LIN {E6POS: X 1455.051, Y -12.200, Z 516.145, A 42.957, B 70.046, C -138.807, E1 0.000, E2 0.0, E3 0.0, E4 0.0, E5 0.0, E6 0.0} C_DIS
;POWDER FEED RATE  =  3.0
;LASER INTENSITY  =  4.0
LIN {E6POS: X 1445.585, Y -2.040, Z 516.145, A 43.012, B 69.711, C -138.813, E1 0.000, E2 0.0, E3 0.0, E4 0.0, E5 0.0, E6 0.0} C_DIS
;POWDER FEED RATE  =  3.0
;LASER INTENSITY  =  4.0
LIN {E6POS: X 1436.083, Y 8.120, Z 516.145, A 43.176, B 69.386, C -138.711, E1 0.000, E2 0.0, E3 0.0, E4 0.0, E5 0.0, E6 0.0} C_DIS
;POWDER FEED RATE  =  3.0
;LASER INTENSITY  =  4.0
LIN {E6POS: X 1426.508, Y 18.280, Z 516.145, A 43.446, B 69.128, C -138.490, E1 0.000, E2 0.0, E3 0.0, E4 0.0, E5 0.0, E6 0.0} C_DIS
;POWDER FEED RATE  =  3.0
;LASER INTENSITY  =  4.0
LIN {E6POS: X 1417.104, Y 28.440, Z 516.393, A 48.821, B 67.331, C -133.472, E1 0.000, E2 0.0, E3 0.0, E4 0.0, E5 0.0, E6 0.0} C_DIS
;POWDER FEED RATE  =  3.0
;LASER INTENSITY  =  4.0
LIN {E6POS: X 1409.237, Y 38.600, Z 518.129, A 60.642, B 62.204, C -122.451, E1 0.000, E2 0.0, E3 0.0, E4 0.0, E5 0.0, E6 0.0} C_DIS
;POWDER FEED RATE  =  3.0
;LASER INTENSITY  =  4.0
LIN {E6POS: X 1404.551, Y 48.760, Z 522.839, A 72.980, B 53.267, C -110.905, E1 0.000, E2 0.0, E3 0.0, E4 0.0, E5 0.0, E6 0.0} C_DIS
;POWDER FEED RATE  =  3.0
;LASER INTENSITY  =  4.0
LIN {E6POS: X 1403.886, Y 58.920, Z 531.268, A 80.416, B 46.343, C -103.137, E1 0.000, E2 0.0, E3 0.0, E4 0.0, E5 0.0, E6 0.0} C_DIS
;POWDER FEED RATE  =  3.0
;LASER INTENSITY  =  4.0
LIN {E6POS: X 1404.867, Y 69.080, Z 541.185, A 83.811, B 46.478, C -98.506, E1 0.000, E2 0.0, E3 0.0, E4 0.0, E5 0.0, E6 0.0} C_DIS
;POWDER FEED RATE  =  3.0
;LASER INTENSITY  =  4.0
LIN {E6POS: X 1404.312, Y 79.240, Z 549.614, A 84.676, B 55.923, C -96.419, E1 0.000, E2 0.0, E3 0.0, E4 0.0, E5 0.0, E6 0.0} C_DIS
;POWDER FEED RATE  =  3.0
;LASER INTENSITY  =  4.0
LIN {E6POS: X 1399.832, Y 89.400, Z 554.324, A 82.280, B 72.116, C -98.107, E1 0.000, E2 0.0, E3 0.0, E4 0.0, E5 0.0, E6 0.0} C_DIS
;POWDER FEED RATE  =  3.0
;LASER INTENSITY  =  4.0
LIN {E6POS: X 1392.206, Y 99.560, Z 556.059, A 70.618, B 83.671, C -109.492, E1 0.000, E2 0.0, E3 0.0, E4 0.0, E5 0.0, E6 0.0} C_DIS
;POWDER FEED RATE  =  3.0
;LASER INTENSITY  =  4.0
LIN {E6POS: X 1383.008, Y 109.720, Z 556.307, A 42.957, B 87.164, C -137.078, E1 0.000, E2 0.0, E3 0.0, E4 0.0, E5 0.0, E6 0.0} C_DIS
;POWDER FEED RATE  =  3.0
;LASER INTENSITY  =  4.0
LIN {E6POS: X 1373.548, Y 119.880, Z 556.307, A 42.957, B 87.129, C -137.079, E1 0.000, E2 0.0, E3 0.0, E4 0.0, E5 0.0, E6 0.0} C_DIS
;POWDER FEED RATE  =  3.0
;LASER INTENSITY  =  4.0
LIN {E6POS: X 1364.087, Y 130.040, Z 556.307, A 42.957, B 87.094, C -137.079, E1 0.000, E2 0.0, E3 0.0, E4 0.0, E5 0.0, E6 0.0} C_DIS
;POWDER FEED RATE  =  3.0
;LASER INTENSITY  =  4.0
LIN {E6POS: X 1354.627, Y 140.200, Z 556.307, A 42.957, B 87.057, C -137.080, E1 0.000, E2 0.0, E3 0.0, E4 0.0, E5 0.0, E6 0.0} C_DIS
;POWDER FEED RATE  =  3.0
;LASER INTENSITY  =  4.0
>>>>>>>>>>>>>>>>>>>>>>>>>>>>POWDER FEED OFF  at=START
>>>>>>>>>>>>>>>>>>>>>>>>>>>>LASER OFF at=START
>>>>>>>>>>>>>>>>>>>>>>>>>>>>GAS SUPPLY OFF  at=START
LIN {E6POS: X 1354.627, Y 140.200, Z 556.307, A 42.957, B 87.057, C -137.080, E1 0.000, E2 0.0, E3 0.0, E4 0.0, E5 0.0, E6 0.0} C_DIS
LIN {E6POS: X 1364.087, Y 130.040, Z 556.307, A 42.957, B 87.094, C -137.079, E1 0.000, E2 0.0, E3 0.0, E4 0.0, E5 0.0, E6 0.0} C_DIS
LIN {E6POS: X 1364.087, Y 130.040, Z 556.307, A 42.957, B 87.094, C -137.079, E1 0.000, E2 0.0, E3 0.0, E4 0.0, E5 0.0, E6 0.0} C_DIS
>>>>>>>>>>>>>>>>>>>>>>>>>>>>GAS SUPPLY ON at=END
>>>>>>>>>>>>>>>>>>>>>>>>>>>>POWDER FEED ON at=END
>>>>>>>>>>>>>>>>>>>>>>>>>>>>LASER ON at=END
LIN {E6POS: X 1459.969, Y -12.200, Z 517.448, A 43.187, B 70.234, C -138.545, E1 0.000, E2 0.0, E3 0.0, E4 0.0, E5 0.0, E6 0.0} C_DIS
;POWDER FEED RATE  =  3.0
;LASER INTENSITY  =  4.0
LIN {E6POS: X 1450.428, Y -2.040, Z 517.448, A 43.224, B 69.979, C -138.554, E1 0.000, E2 0.0, E3 0.0, E4 0.0, E5 0.0, E6 0.0} C_DIS
;POWDER FEED RATE  =  3.0
;LASER INTENSITY  =  4.0
LIN {E6POS: X 1440.864, Y 8.120, Z 517.448, A 43.333, B 69.736, C -138.490, E1 0.000, E2 0.0, E3 0.0, E4 0.0, E5 0.0, E6 0.0} C_DIS
;POWDER FEED RATE  =  3.0
;LASER INTENSITY  =  4.0
LIN {E6POS: X 1431.250, Y 18.280, Z 517.448, A 43.513, B 69.549, C -138.345, E1 0.000, E2 0.0, E3 0.0, E4 0.0, E5 0.0, E6 0.0} C_DIS
;POWDER FEED RATE  =  3.0
;LASER INTENSITY  =  4.0
LIN {E6POS: X 1421.855, Y 28.440, Z 517.689, A 48.669, B 67.874, C -133.513, E1 0.000, E2 0.0, E3 0.0, E4 0.0, E5 0.0, E6 0.0} C_DIS
;POWDER FEED RATE  =  3.0
;LASER INTENSITY  =  4.0
LIN {E6POS: X 1414.112, Y 38.600, Z 519.378, A 60.307, B 63.006, C -122.617, E1 0.000, E2 0.0, E3 0.0, E4 0.0, E5 0.0, E6 0.0} C_DIS
;POWDER FEED RATE  =  3.0
;LASER INTENSITY  =  4.0
LIN {E6POS: X 1409.744, Y 48.760, Z 523.963, A 72.750, B 54.338, C -110.916, E1 0.000, E2 0.0, E3 0.0, E4 0.0, E5 0.0, E6 0.0} C_DIS
;POWDER FEED RATE  =  3.0
;LASER INTENSITY  =  4.0
LIN {E6POS: X 1409.627, Y 58.920, Z 532.166, A 80.409, B 47.407, C -102.927, E1 0.000, E2 0.0, E3 0.0, E4 0.0, E5 0.0, E6 0.0} C_DIS
;POWDER FEED RATE  =  3.0
;LASER INTENSITY  =  4.0
LIN {E6POS: X 1411.234, Y 69.080, Z 541.818, A 83.997, B 47.432, C -98.125, E1 0.000, E2 0.0, E3 0.0, E4 0.0, E5 0.0, E6 0.0} C_DIS
;POWDER FEED RATE  =  3.0
;LASER INTENSITY  =  4.0
LIN {E6POS: X 1411.190, Y 79.240, Z 550.021, A 85.122, B 56.795, C -95.824, E1 0.000, E2 0.0, E3 0.0, E4 0.0, E5 0.0, E6 0.0} C_DIS
;POWDER FEED RATE  =  3.0
;LASER INTENSITY  =  4.0
LIN {E6POS: X 1406.961, Y 89.400, Z 554.606, A 83.358, B 72.840, C -96.948, E1 0.000, E2 0.0, E3 0.0, E4 0.0, E5 0.0, E6 0.0} C_DIS
;POWDER FEED RATE  =  3.0
;LASER INTENSITY  =  4.0
LIN {E6POS: X 1399.379, Y 99.560, Z 556.295, A 73.249, B 84.276, C -106.830, E1 0.000, E2 0.0, E3 0.0, E4 0.0, E5 0.0, E6 0.0} C_DIS
;POWDER FEED RATE  =  3.0
;LASER INTENSITY  =  4.0
LIN {E6POS: X 1390.122, Y 109.720, Z 556.536, A 43.187, B 87.789, C -136.834, E1 0.000, E2 0.0, E3 0.0, E4 0.0, E5 0.0, E6 0.0} C_DIS
;POWDER FEED RATE  =  3.0
;LASER INTENSITY  =  4.0
LIN {E6POS: X 1380.585, Y 119.880, Z 556.536, A 43.187, B 87.769, C -136.834, E1 0.000, E2 0.0, E3 0.0, E4 0.0, E5 0.0, E6 0.0} C_DIS
;POWDER FEED RATE  =  3.0
;LASER INTENSITY  =  4.0
LIN {E6POS: X 1371.049, Y 130.040, Z 556.536, A 43.187, B 87.747, C -136.835, E1 0.000, E2 0.0, E3 0.0, E4 0.0, E5 0.0, E6 0.0} C_DIS
;POWDER FEED RATE  =  3.0
;LASER INTENSITY  =  4.0
LIN {E6POS: X 1361.512, Y 140.200, Z 556.536, A 43.187, B 87.725, C -136.835, E1 0.000, E2 0.0, E3 0.0, E4 0.0, E5 0.0, E6 0.0} C_DIS
;POWDER FEED RATE  =  3.0
;LASER INTENSITY  =  4.0
>>>>>>>>>>>>>>>>>>>>>>>>>>>>POWDER FEED OFF  at=START
>>>>>>>>>>>>>>>>>>>>>>>>>>>>LASER OFF at=START
>>>>>>>>>>>>>>>>>>>>>>>>>>>>GAS SUPPLY OFF  at=START
LIN {E6POS: X 1361.512, Y 140.200, Z 556.536, A 43.187, B 87.725, C -136.835, E1 0.000, E2 0.0, E3 0.0, E4 0.0, E5 0.0, E6 0.0} C_DIS
LIN {E6POS: X 1371.049, Y 130.040, Z 556.536, A 43.187, B 87.747, C -136.835, E1 0.000, E2 0.0, E3 0.0, E4 0.0, E5 0.0, E6 0.0} C_DIS
LIN {E6POS: X 1371.049, Y 130.040, Z 556.536, A 43.187, B 87.747, C -136.835, E1 0.000, E2 0.0, E3 0.0, E4 0.0, E5 0.0, E6 0.0} C_DIS
>>>>>>>>>>>>>>>>>>>>>>>>>>>>GAS SUPPLY ON at=END
>>>>>>>>>>>>>>>>>>>>>>>>>>>>POWDER FEED ON at=END
>>>>>>>>>>>>>>>>>>>>>>>>>>>>LASER ON at=END
LIN {E6POS: X 1464.867, Y -12.200, Z 518.698, A 43.359, B 71.280, C -138.192, E1 0.000, E2 0.0, E3 0.0, E4 0.0, E5 0.0, E6 0.0} C_DIS
;POWDER FEED RATE  =  3.0
;LASER INTENSITY  =  4.0
LIN {E6POS: X 1455.270, Y -2.040, Z 518.698, A 43.382, B 71.104, C -138.200, E1 0.000, E2 0.0, E3 0.0, E4 0.0, E5 0.0, E6 0.0} C_DIS
;POWDER FEED RATE  =  3.0
;LASER INTENSITY  =  4.0
LIN {E6POS: X 1445.658, Y 8.120, Z 518.698, A 43.450, B 70.939, C -138.160, E1 0.000, E2 0.0, E3 0.0, E4 0.0, E5 0.0, E6 0.0} C_DIS
;POWDER FEED RATE  =  3.0
;LASER INTENSITY  =  4.0
LIN {E6POS: X 1436.016, Y 18.280, Z 518.698, A 43.563, B 70.815, C -138.068, E1 0.000, E2 0.0, E3 0.0, E4 0.0, E5 0.0, E6 0.0} C_DIS
;POWDER FEED RATE  =  3.0
;LASER INTENSITY  =  4.0
LIN {E6POS: X 1426.630, Y 28.440, Z 518.932, A 48.837, B 69.183, C -133.087, E1 0.000, E2 0.0, E3 0.0, E4 0.0, E5 0.0, E6 0.0} C_DIS
;POWDER FEED RATE  =  3.0
;LASER INTENSITY  =  4.0
LIN {E6POS: X 1419.000, Y 38.600, Z 520.575, A 60.708, B 64.304, C -121.904, E1 0.000, E2 0.0, E3 0.0, E4 0.0, E5 0.0, E6 0.0} C_DIS
;POWDER FEED RATE  =  3.0
;LASER INTENSITY  =  4.0
LIN {E6POS: X 1414.928, Y 48.760, Z 525.033, A 73.166, B 55.549, C -110.150, E1 0.000, E2 0.0, E3 0.0, E4 0.0, E5 0.0, E6 0.0} C_DIS
;POWDER FEED RATE  =  3.0
;LASER INTENSITY  =  4.0
LIN {E6POS: X 1415.321, Y 58.920, Z 533.010, A 80.752, B 48.468, C -102.271, E1 0.000, E2 0.0, E3 0.0, E4 0.0, E5 0.0, E6 0.0} C_DIS
;POWDER FEED RATE  =  3.0
;LASER INTENSITY  =  4.0
LIN {E6POS: X 1417.517, Y 69.080, Z 542.395, A 84.350, B 48.378, C -97.539, E1 0.000, E2 0.0, E3 0.0, E4 0.0, E5 0.0, E6 0.0} C_DIS
;POWDER FEED RATE  =  3.0
;LASER INTENSITY  =  4.0
LIN {E6POS: X 1417.956, Y 79.240, Z 550.373, A 85.638, B 57.664, C -95.159, E1 0.000, E2 0.0, E3 0.0, E4 0.0, E5 0.0, E6 0.0} C_DIS
;POWDER FEED RATE  =  3.0
;LASER INTENSITY  =  4.0
LIN {E6POS: X 1413.970, Y 89.400, Z 554.831, A 84.454, B 73.537, C -95.781, E1 0.000, E2 0.0, E3 0.0, E4 0.0, E5 0.0, E6 0.0} C_DIS
;POWDER FEED RATE  =  3.0
;LASER INTENSITY  =  4.0
LIN {E6POS: X 1406.442, Y 99.560, Z 556.473, A 76.097, B 84.824, C -103.958, E1 0.000, E2 0.0, E3 0.0, E4 0.0, E5 0.0, E6 0.0} C_DIS
;POWDER FEED RATE  =  3.0
;LASER INTENSITY  =  4.0
LIN {E6POS: X 1397.144, Y 109.720, Z 556.708, A 43.359, B 88.351, C -136.653, E1 0.000, E2 0.0, E3 0.0, E4 0.0, E5 0.0, E6 0.0} C_DIS
;POWDER FEED RATE  =  3.0
;LASER INTENSITY  =  4.0
LIN {E6POS: X 1387.550, Y 119.880, Z 556.708, A 43.359, B 88.339, C -136.653, E1 0.000, E2 0.0, E3 0.0, E4 0.0, E5 0.0, E6 0.0} C_DIS
;POWDER FEED RATE  =  3.0
;LASER INTENSITY  =  4.0
LIN {E6POS: X 1377.956, Y 130.040, Z 556.708, A 43.359, B 88.328, C -136.653, E1 0.000, E2 0.0, E3 0.0, E4 0.0, E5 0.0, E6 0.0} C_DIS
;POWDER FEED RATE  =  3.0
;LASER INTENSITY  =  4.0
LIN {E6POS: X 1368.361, Y 140.200, Z 556.708, A 43.359, B 88.316, C -136.653, E1 0.000, E2 0.0, E3 0.0, E4 0.0, E5 0.0, E6 0.0} C_DIS
;POWDER FEED RATE  =  3.0
;LASER INTENSITY  =  4.0
>>>>>>>>>>>>>>>>>>>>>>>>>>>>POWDER FEED OFF  at=START
>>>>>>>>>>>>>>>>>>>>>>>>>>>>LASER OFF at=START
>>>>>>>>>>>>>>>>>>>>>>>>>>>>GAS SUPPLY OFF  at=START
LIN {E6POS: X 1368.361, Y 140.200, Z 556.708, A 43.359, B 88.316, C -136.653, E1 0.000, E2 0.0, E3 0.0, E4 0.0, E5 0.0, E6 0.0} C_DIS
LIN {E6POS: X 1377.956, Y 130.040, Z 556.708, A 43.359, B 88.328, C -136.653, E1 0.000, E2 0.0, E3 0.0, E4 0.0, E5 0.0, E6 0.0} C_DIS
LIN {E6POS: X 1377.956, Y 130.040, Z 556.708, A 43.359, B 88.328, C -136.653, E1 0.000, E2 0.0, E3 0.0, E4 0.0, E5 0.0, E6 0.0} C_DIS
>>>>>>>>>>>>>>>>>>>>>>>>>>>>GAS SUPPLY ON at=END
>>>>>>>>>>>>>>>>>>>>>>>>>>>>POWDER FEED ON at=END
>>>>>>>>>>>>>>>>>>>>>>>>>>>>LASER ON at=END
LIN {E6POS: X 1469.825, Y -12.200, Z 519.857, A 43.481, B 73.154, C -137.772, E1 0.000, E2 0.0, E3 0.0, E4 0.0, E5 0.0, E6 0.0} C_DIS
;POWDER FEED RATE  =  3.0
;LASER INTENSITY  =  4.0
LIN {E6POS: X 1460.188, Y -2.040, Z 519.857, A 43.494, B 73.045, C -137.775, E1 0.000, E2 0.0, E3 0.0, E4 0.0, E5 0.0, E6 0.0} C_DIS
;POWDER FEED RATE  =  3.0
;LASER INTENSITY  =  4.0
LIN {E6POS: X 1450.543, Y 8.120, Z 519.857, A 43.534, B 72.945, C -137.751, E1 0.000, E2 0.0, E3 0.0, E4 0.0, E5 0.0, E6 0.0} C_DIS
;POWDER FEED RATE  =  3.0
;LASER INTENSITY  =  4.0
LIN {E6POS: X 1440.880, Y 18.280, Z 519.857, A 43.599, B 72.872, C -137.697, E1 0.000, E2 0.0, E3 0.0, E4 0.0, E5 0.0, E6 0.0} C_DIS
;POWDER FEED RATE  =  3.0
;LASER INTENSITY  =  4.0
LIN {E6POS: X 1431.504, Y 28.440, Z 520.085, A 49.405, B 71.202, C -132.153, E1 0.000, E2 0.0, E3 0.0, E4 0.0, E5 0.0, E6 0.0} C_DIS
;POWDER FEED RATE  =  3.0
;LASER INTENSITY  =  4.0
LIN {E6POS: X 1423.975, Y 38.600, Z 521.683, A 61.989, B 66.034, C -120.206, E1 0.000, E2 0.0, E3 0.0, E4 0.0, E5 0.0, E6 0.0} C_DIS
;POWDER FEED RATE  =  3.0
;LASER INTENSITY  =  4.0
LIN {E6POS: X 1420.168, Y 48.760, Z 526.019, A 74.316, B 56.821, C -108.546, E1 0.000, E2 0.0, E3 0.0, E4 0.0, E5 0.0, E6 0.0} C_DIS
;POWDER FEED RATE  =  3.0
;LASER INTENSITY  =  4.0
LIN {E6POS: X 1421.025, Y 58.920, Z 533.779, A 81.485, B 49.455, C -101.145, E1 0.000, E2 0.0, E3 0.0, E4 0.0, E5 0.0, E6 0.0} C_DIS
;POWDER FEED RATE  =  3.0
;LASER INTENSITY  =  4.0
LIN {E6POS: X 1423.755, Y 69.080, Z 542.909, A 84.887, B 49.265, C -96.735, E1 0.000, E2 0.0, E3 0.0, E4 0.0, E5 0.0, E6 0.0} C_DIS
;POWDER FEED RATE  =  3.0
;LASER INTENSITY  =  4.0
LIN {E6POS: X 1424.638, Y 79.240, Z 550.669, A 86.227, B 58.494, C -94.423, E1 0.000, E2 0.0, E3 0.0, E4 0.0, E5 0.0, E6 0.0} C_DIS
;POWDER FEED RATE  =  3.0
;LASER INTENSITY  =  4.0
LIN {E6POS: X 1420.881, Y 89.400, Z 555.005, A 85.552, B 74.187, C -94.622, E1 0.000, E2 0.0, E3 0.0, E4 0.0, E5 0.0, E6 0.0} C_DIS
;POWDER FEED RATE  =  3.0
;LASER INTENSITY  =  4.0
LIN {E6POS: X 1413.412, Y 99.560, Z 556.603, A 79.104, B 85.302, C -100.932, E1 0.000, E2 0.0, E3 0.0, E4 0.0, E5 0.0, E6 0.0} C_DIS
;POWDER FEED RATE  =  3.0
;LASER INTENSITY  =  4.0
LIN {E6POS: X 1404.086, Y 109.720, Z 556.831, A 43.481, B 88.840, C -136.525, E1 0.000, E2 0.0, E3 0.0, E4 0.0, E5 0.0, E6 0.0} C_DIS
;POWDER FEED RATE  =  3.0
;LASER INTENSITY  =  4.0
LIN {E6POS: X 1394.451, Y 119.880, Z 556.831, A 43.481, B 88.835, C -136.525, E1 0.000, E2 0.0, E3 0.0, E4 0.0, E5 0.0, E6 0.0} C_DIS
;POWDER FEED RATE  =  3.0
;LASER INTENSITY  =  4.0
LIN {E6POS: X 1384.816, Y 130.040, Z 556.831, A 43.481, B 88.829, C -136.525, E1 0.000, E2 0.0, E3 0.0, E4 0.0, E5 0.0, E6 0.0} C_DIS
;POWDER FEED RATE  =  3.0
;LASER INTENSITY  =  4.0
LIN {E6POS: X 1375.181, Y 140.200, Z 556.831, A 43.481, B 88.823, C -136.525, E1 0.000, E2 0.0, E3 0.0, E4 0.0, E5 0.0, E6 0.0} C_DIS
;POWDER FEED RATE  =  3.0
;LASER INTENSITY  =  4.0
>>>>>>>>>>>>>>>>>>>>>>>>>>>>POWDER FEED OFF  at=START
>>>>>>>>>>>>>>>>>>>>>>>>>>>>LASER OFF at=START
>>>>>>>>>>>>>>>>>>>>>>>>>>>>GAS SUPPLY OFF  at=START
LIN {E6POS: X 1375.181, Y 140.200, Z 556.831, A 43.481, B 88.823, C -136.525, E1 0.000, E2 0.0, E3 0.0, E4 0.0, E5 0.0, E6 0.0} C_DIS
LIN {E6POS: X 1384.816, Y 130.040, Z 556.831, A 43.481, B 88.829, C -136.525, E1 0.000, E2 0.0, E3 0.0, E4 0.0, E5 0.0, E6 0.0} C_DIS
LIN {E6POS: X 1384.816, Y 130.040, Z 556.831, A 43.481, B 88.829, C -136.525, E1 0.000, E2 0.0, E3 0.0, E4 0.0, E5 0.0, E6 0.0} C_DIS
>>>>>>>>>>>>>>>>>>>>>>>>>>>>GAS SUPPLY ON at=END
>>>>>>>>>>>>>>>>>>>>>>>>>>>>POWDER FEED ON at=END
>>>>>>>>>>>>>>>>>>>>>>>>>>>>LASER ON at=END
LIN {E6POS: X 1474.925, Y -12.200, Z 520.889, A 43.563, B 75.759, C -137.329, E1 0.000, E2 0.0, E3 0.0, E4 0.0, E5 0.0, E6 0.0} C_DIS
;POWDER FEED RATE  =  3.0
;LASER INTENSITY  =  4.0
LIN {E6POS: X 1465.262, Y -2.040, Z 520.889, A 43.570, B 75.702, C -137.330, E1 0.000, E2 0.0, E3 0.0, E4 0.0, E5 0.0, E6 0.0} C_DIS
;POWDER FEED RATE  =  3.0
;LASER INTENSITY  =  4.0
LIN {E6POS: X 1455.594, Y 8.120, Z 520.889, A 43.590, B 75.650, C -137.316, E1 0.000, E2 0.0, E3 0.0, E4 0.0, E5 0.0, E6 0.0} C_DIS
;POWDER FEED RATE  =  3.0
;LASER INTENSITY  =  4.0
LIN {E6POS: X 1445.917, Y 18.280, Z 520.889, A 43.623, B 75.613, C -137.287, E1 0.000, E2 0.0, E3 0.0, E4 0.0, E5 0.0, E6 0.0} C_DIS
;POWDER FEED RATE  =  3.0
;LASER INTENSITY  =  4.0
LIN {E6POS: X 1436.550, Y 28.440, Z 521.112, A 50.550, B 73.825, C -130.590, E1 0.000, E2 0.0, E3 0.0, E4 0.0, E5 0.0, E6 0.0} C_DIS
;POWDER FEED RATE  =  3.0
;LASER INTENSITY  =  4.0
LIN {E6POS: X 1429.109, Y 38.600, Z 522.668, A 64.346, B 68.087, C -117.369, E1 0.000, E2 0.0, E3 0.0, E4 0.0, E5 0.0, E6 0.0} C_DIS
;POWDER FEED RATE  =  3.0
;LASER INTENSITY  =  4.0
LIN {E6POS: X 1425.532, Y 48.760, Z 526.893, A 76.244, B 58.061, C -106.091, E1 0.000, E2 0.0, E3 0.0, E4 0.0, E5 0.0, E6 0.0} C_DIS
;POWDER FEED RATE  =  3.0
;LASER INTENSITY  =  4.0
LIN {E6POS: X 1426.793, Y 58.920, Z 534.454, A 82.621, B 50.297, C -99.555, E1 0.000, E2 0.0, E3 0.0, E4 0.0, E5 0.0, E6 0.0} C_DIS
;POWDER FEED RATE  =  3.0
;LASER INTENSITY  =  4.0
LIN {E6POS: X 1429.992, Y 69.080, Z 543.349, A 85.614, B 50.041, C -95.714, E1 0.000, E2 0.0, E3 0.0, E4 0.0, E5 0.0, E6 0.0} C_DIS
;POWDER FEED RATE  =  3.0
;LASER INTENSITY  =  4.0
LIN {E6POS: X 1431.266, Y 79.240, Z 550.909, A 86.889, B 59.250, C -93.619, E1 0.000, E2 0.0, E3 0.0, E4 0.0, E5 0.0, E6 0.0} C_DIS
;POWDER FEED RATE  =  3.0
;LASER INTENSITY  =  4.0
LIN {E6POS: X 1427.715, Y 89.400, Z 555.134, A 86.628, B 74.770, C -93.495, E1 0.000, E2 0.0, E3 0.0, E4 0.0, E5 0.0, E6 0.0} C_DIS
;POWDER FEED RATE  =  3.0
;LASER INTENSITY  =  4.0
LIN {E6POS: X 1420.304, Y 99.560, Z 556.691, A 82.147, B 85.702, C -97.875, E1 0.000, E2 0.0, E3 0.0, E4 0.0, E5 0.0, E6 0.0} C_DIS
;POWDER FEED RATE  =  3.0
;LASER INTENSITY  =  4.0
LIN {E6POS: X 1410.963, Y 109.720, Z 556.913, A 43.563, B 89.250, C -136.439, E1 0.000, E2 0.0, E3 0.0, E4 0.0, E5 0.0, E6 0.0} C_DIS
;POWDER FEED RATE  =  3.0
;LASER INTENSITY  =  4.0
LIN {E6POS: X 1401.300, Y 119.880, Z 556.913, A 43.563, B 89.248, C -136.439, E1 0.000, E2 0.0, E3 0.0, E4 0.0, E5 0.0, E6 0.0} C_DIS
;POWDER FEED RATE  =  3.0
;LASER INTENSITY  =  4.0
LIN {E6POS: X 1391.638, Y 130.040, Z 556.913, A 43.563, B 89.246, C -136.439, E1 0.000, E2 0.0, E3 0.0, E4 0.0, E5 0.0, E6 0.0} C_DIS
;POWDER FEED RATE  =  3.0
;LASER INTENSITY  =  4.0
LIN {E6POS: X 1381.975, Y 140.200, Z 556.913, A 43.563, B 89.243, C -136.439, E1 0.000, E2 0.0, E3 0.0, E4 0.0, E5 0.0, E6 0.0} C_DIS
;POWDER FEED RATE  =  3.0
;LASER INTENSITY  =  4.0
>>>>>>>>>>>>>>>>>>>>>>>>>>>>POWDER FEED OFF  at=START
>>>>>>>>>>>>>>>>>>>>>>>>>>>>LASER OFF at=START
>>>>>>>>>>>>>>>>>>>>>>>>>>>>GAS SUPPLY OFF  at=START
LIN {E6POS: X 1381.975, Y 140.200, Z 556.913, A 43.563, B 89.243, C -136.439, E1 0.000, E2 0.0, E3 0.0, E4 0.0, E5 0.0, E6 0.0} C_DIS
LIN {E6POS: X 1391.638, Y 130.040, Z 556.913, A 43.563, B 89.246, C -136.439, E1 0.000, E2 0.0, E3 0.0, E4 0.0, E5 0.0, E6 0.0} C_DIS
LIN {E6POS: X 1391.638, Y 130.040, Z 556.913, A 43.563, B 89.246, C -136.439, E1 0.000, E2 0.0, E3 0.0, E4 0.0, E5 0.0, E6 0.0} C_DIS
>>>>>>>>>>>>>>>>>>>>>>>>>>>>GAS SUPPLY ON at=END
>>>>>>>>>>>>>>>>>>>>>>>>>>>>POWDER FEED ON at=END
>>>>>>>>>>>>>>>>>>>>>>>>>>>>LASER ON at=END
LIN {E6POS: X 1480.249, Y -12.200, Z 521.757, A 43.613, B 78.943, C -136.923, E1 0.000, E2 0.0, E3 0.0, E4 0.0, E5 0.0, E6 0.0} C_DIS
;POWDER FEED RATE  =  3.0
;LASER INTENSITY  =  4.0
LIN {E6POS: X 1470.570, Y -2.040, Z 521.757, A 43.615, B 78.919, C -136.923, E1 0.000, E2 0.0, E3 0.0, E4 0.0, E5 0.0, E6 0.0} C_DIS
;POWDER FEED RATE  =  3.0
;LASER INTENSITY  =  4.0
LIN {E6POS: X 1460.888, Y 8.120, Z 521.757, A 43.624, B 78.898, C -136.917, E1 0.000, E2 0.0, E3 0.0, E4 0.0, E5 0.0, E6 0.0} C_DIS
;POWDER FEED RATE  =  3.0
;LASER INTENSITY  =  4.0
LIN {E6POS: X 1451.202, Y 18.280, Z 521.757, A 43.638, B 78.883, C -136.904, E1 0.000, E2 0.0, E3 0.0, E4 0.0, E5 0.0, E6 0.0} C_DIS
;POWDER FEED RATE  =  3.0
;LASER INTENSITY  =  4.0
LIN {E6POS: X 1441.844, Y 28.440, Z 521.974, A 52.654, B 76.899, C -128.077, E1 0.000, E2 0.0, E3 0.0, E4 0.0, E5 0.0, E6 0.0} C_DIS
;POWDER FEED RATE  =  3.0
;LASER INTENSITY  =  4.0
LIN {E6POS: X 1434.474, Y 38.600, Z 523.495, A 68.044, B 70.311, C -113.179, E1 0.000, E2 0.0, E3 0.0, E4 0.0, E5 0.0, E6 0.0} C_DIS
;POWDER FEED RATE  =  3.0
;LASER INTENSITY  =  4.0
LIN {E6POS: X 1431.087, Y 48.760, Z 527.625, A 78.927, B 59.167, C -102.839, E1 0.000, E2 0.0, E3 0.0, E4 0.0, E5 0.0, E6 0.0} C_DIS
;POWDER FEED RATE  =  3.0
;LASER INTENSITY  =  4.0
LIN {E6POS: X 1432.681, Y 58.920, Z 535.014, A 84.127, B 50.928, C -97.547, E1 0.000, E2 0.0, E3 0.0, E4 0.0, E5 0.0, E6 0.0} C_DIS
;POWDER FEED RATE  =  3.0
;LASER INTENSITY  =  4.0
LIN {E6POS: X 1436.269, Y 69.080, Z 543.707, A 86.522, B 50.656, C -94.493, E1 0.000, E2 0.0, E3 0.0, E4 0.0, E5 0.0, E6 0.0} C_DIS
;POWDER FEED RATE  =  3.0
;LASER INTENSITY  =  4.0
LIN {E6POS: X 1437.868, Y 79.240, Z 551.096, A 87.615, B 59.897, C -92.757, E1 0.000, E2 0.0, E3 0.0, E4 0.0, E5 0.0, E6 0.0} C_DIS
;POWDER FEED RATE  =  3.0
;LASER INTENSITY  =  4.0
LIN {E6POS: X 1434.492, Y 89.400, Z 555.225, A 87.648, B 75.267, C -92.431, E1 0.000, E2 0.0, E3 0.0, E4 0.0, E5 0.0, E6 0.0} C_DIS
;POWDER FEED RATE  =  3.0
;LASER INTENSITY  =  4.0
LIN {E6POS: X 1427.135, Y 99.560, Z 556.746, A 85.025, B 86.019, C -94.987, E1 0.000, E2 0.0, E3 0.0, E4 0.0, E5 0.0, E6 0.0} C_DIS
;POWDER FEED RATE  =  3.0
;LASER INTENSITY  =  4.0
LIN {E6POS: X 1417.787, Y 109.720, Z 556.963, A 43.613, B 89.575, C -136.388, E1 0.000, E2 0.0, E3 0.0, E4 0.0, E5 0.0, E6 0.0} C_DIS
;POWDER FEED RATE  =  3.0
;LASER INTENSITY  =  4.0
LIN {E6POS: X 1408.108, Y 119.880, Z 556.963, A 43.613, B 89.574, C -136.388, E1 0.000, E2 0.0, E3 0.0, E4 0.0, E5 0.0, E6 0.0} C_DIS
;POWDER FEED RATE  =  3.0
;LASER INTENSITY  =  4.0
LIN {E6POS: X 1398.428, Y 130.040, Z 556.963, A 43.613, B 89.574, C -136.388, E1 0.000, E2 0.0, E3 0.0, E4 0.0, E5 0.0, E6 0.0} C_DIS
;POWDER FEED RATE  =  3.0
;LASER INTENSITY  =  4.0
LIN {E6POS: X 1388.749, Y 140.200, Z 556.963, A 43.613, B 89.573, C -136.388, E1 0.000, E2 0.0, E3 0.0, E4 0.0, E5 0.0, E6 0.0} C_DIS
;POWDER FEED RATE  =  3.0
;LASER INTENSITY  =  4.0
>>>>>>>>>>>>>>>>>>>>>>>>>>>>POWDER FEED OFF  at=START
>>>>>>>>>>>>>>>>>>>>>>>>>>>>LASER OFF at=START
>>>>>>>>>>>>>>>>>>>>>>>>>>>>GAS SUPPLY OFF  at=START
LIN {E6POS: X 1388.749, Y 140.200, Z 556.963, A 43.613, B 89.573, C -136.388, E1 0.000, E2 0.0, E3 0.0, E4 0.0, E5 0.0, E6 0.0} C_DIS
LIN {E6POS: X 1398.428, Y 130.040, Z 556.963, A 43.613, B 89.574, C -136.388, E1 0.000, E2 0.0, E3 0.0, E4 0.0, E5 0.0, E6 0.0} C_DIS
LIN {E6POS: X 1398.428, Y 130.040, Z 556.963, A 43.613, B 89.574, C -136.388, E1 0.000, E2 0.0, E3 0.0, E4 0.0, E5 0.0, E6 0.0} C_DIS
>>>>>>>>>>>>>>>>>>>>>>>>>>>>GAS SUPPLY ON at=END
>>>>>>>>>>>>>>>>>>>>>>>>>>>>POWDER FEED ON at=END
>>>>>>>>>>>>>>>>>>>>>>>>>>>>LASER ON at=END
LIN {E6POS: X 1485.878, Y -12.200, Z 522.423, A 43.638, B 82.512, C -136.607, E1 0.000, E2 0.0, E3 0.0, E4 0.0, E5 0.0, E6 0.0} C_DIS
;POWDER FEED RATE  =  3.0
;LASER INTENSITY  =  4.0
LIN {E6POS: X 1476.190, Y -2.040, Z 522.423, A 43.639, B 82.505, C -136.607, E1 0.000, E2 0.0, E3 0.0, E4 0.0, E5 0.0, E6 0.0} C_DIS
;POWDER FEED RATE  =  3.0
;LASER INTENSITY  =  4.0
LIN {E6POS: X 1466.501, Y 8.120, Z 522.423, A 43.641, B 82.499, C -136.605, E1 0.000, E2 0.0, E3 0.0, E4 0.0, E5 0.0, E6 0.0} C_DIS
;POWDER FEED RATE  =  3.0
;LASER INTENSITY  =  4.0
LIN {E6POS: X 1456.811, Y 18.280, Z 522.423, A 43.645, B 82.495, C -136.601, E1 0.000, E2 0.0, E3 0.0, E4 0.0, E5 0.0, E6 0.0} C_DIS
;POWDER FEED RATE  =  3.0
;LASER INTENSITY  =  4.0
LIN {E6POS: X 1447.460, Y 28.440, Z 522.636, A 56.647, B 80.231, C -123.739, E1 0.000, E2 0.0, E3 0.0, E4 0.0, E5 0.0, E6 0.0} C_DIS
;POWDER FEED RATE  =  3.0
;LASER INTENSITY  =  4.0
LIN {E6POS: X 1440.143, Y 38.600, Z 524.130, A 73.396, B 72.519, C -107.361, E1 0.000, E2 0.0, E3 0.0, E4 0.0, E5 0.0, E6 0.0} C_DIS
;POWDER FEED RATE  =  3.0
;LASER INTENSITY  =  4.0
LIN {E6POS: X 1436.898, Y 48.760, Z 528.184, A 82.254, B 60.043, C -98.922, E1 0.000, E2 0.0, E3 0.0, E4 0.0, E5 0.0, E6 0.0} C_DIS
;POWDER FEED RATE  =  3.0
;LASER INTENSITY  =  4.0
LIN {E6POS: X 1438.744, Y 58.920, Z 535.438, A 85.934, B 51.296, C -95.205, E1 0.000, E2 0.0, E3 0.0, E4 0.0, E5 0.0, E6 0.0} C_DIS
;POWDER FEED RATE  =  3.0
;LASER INTENSITY  =  4.0
LIN {E6POS: X 1442.627, Y 69.080, Z 543.973, A 87.587, B 51.065, C -93.101, E1 0.000, E2 0.0, E3 0.0, E4 0.0, E5 0.0, E6 0.0} C_DIS
;POWDER FEED RATE  =  3.0
;LASER INTENSITY  =  4.0
LIN {E6POS: X 1444.475, Y 79.240, Z 551.228, A 88.390, B 60.400, C -91.851, E1 0.000, E2 0.0, E3 0.0, E4 0.0, E5 0.0, E6 0.0} C_DIS
;POWDER FEED RATE  =  3.0
;LASER INTENSITY  =  4.0
LIN {E6POS: X 1441.234, Y 89.400, Z 555.282, A 88.577, B 75.662, C -91.468, E1 0.000, E2 0.0, E3 0.0, E4 0.0, E5 0.0, E6 0.0} C_DIS
;POWDER FEED RATE  =  3.0
;LASER INTENSITY  =  4.0
LIN {E6POS: X 1433.921, Y 99.560, Z 556.776, A 87.475, B 86.251, C -92.531, E1 0.000, E2 0.0, E3 0.0, E4 0.0, E5 0.0, E6 0.0} C_DIS
;POWDER FEED RATE  =  3.0
;LASER INTENSITY  =  4.0
LIN {E6POS: X 1424.572, Y 109.720, Z 556.989, A 43.638, B 89.810, C -136.362, E1 0.000, E2 0.0, E3 0.0, E4 0.0, E5 0.0, E6 0.0} C_DIS
;POWDER FEED RATE  =  3.0
;LASER INTENSITY  =  4.0
LIN {E6POS: X 1414.884, Y 119.880, Z 556.989, A 43.638, B 89.810, C -136.362, E1 0.000, E2 0.0, E3 0.0, E4 0.0, E5 0.0, E6 0.0} C_DIS
;POWDER FEED RATE  =  3.0
;LASER INTENSITY  =  4.0
LIN {E6POS: X 1405.196, Y 130.040, Z 556.989, A 43.638, B 89.810, C -136.362, E1 0.000, E2 0.0, E3 0.0, E4 0.0, E5 0.0, E6 0.0} C_DIS
;POWDER FEED RATE  =  3.0
;LASER INTENSITY  =  4.0
LIN {E6POS: X 1395.508, Y 140.200, Z 556.989, A 43.638, B 89.810, C -136.362, E1 0.000, E2 0.0, E3 0.0, E4 0.0, E5 0.0, E6 0.0} C_DIS
;POWDER FEED RATE  =  3.0
;LASER INTENSITY  =  4.0
>>>>>>>>>>>>>>>>>>>>>>>>>>>>POWDER FEED OFF  at=START
>>>>>>>>>>>>>>>>>>>>>>>>>>>>LASER OFF at=START
>>>>>>>>>>>>>>>>>>>>>>>>>>>>GAS SUPPLY OFF  at=START
LIN {E6POS: X 1395.508, Y 140.200, Z 556.989, A 43.638, B 89.810, C -136.362, E1 0.000, E2 0.0, E3 0.0, E4 0.0, E5 0.0, E6 0.0} C_DIS
LIN {E6POS: X 1405.196, Y 130.040, Z 556.989, A 43.638, B 89.810, C -136.362, E1 0.000, E2 0.0, E3 0.0, E4 0.0, E5 0.0, E6 0.0} C_DIS
LIN {E6POS: X 1405.196, Y 130.040, Z 556.989, A 43.638, B 89.810, C -136.362, E1 0.000, E2 0.0, E3 0.0, E4 0.0, E5 0.0, E6 0.0} C_DIS
>>>>>>>>>>>>>>>>>>>>>>>>>>>>GAS SUPPLY ON at=END
>>>>>>>>>>>>>>>>>>>>>>>>>>>>POWDER FEED ON at=END
>>>>>>>>>>>>>>>>>>>>>>>>>>>>LASER ON at=END
LIN {E6POS: X 1491.893, Y -12.200, Z 522.849, A 43.647, B 86.261, C -136.414, E1 0.000, E2 0.0, E3 0.0, E4 0.0, E5 0.0, E6 0.0} C_DIS
;POWDER FEED RATE  =  3.0
;LASER INTENSITY  =  4.0
LIN {E6POS: X 1482.202, Y -2.040, Z 522.849, A 43.647, B 86.260, C -136.414, E1 0.000, E2 0.0, E3 0.0, E4 0.0, E5 0.0, E6 0.0} C_DIS
;POWDER FEED RATE  =  3.0
;LASER INTENSITY  =  4.0
LIN {E6POS: X 1472.510, Y 8.120, Z 522.849, A 43.648, B 86.259, C -136.413, E1 0.000, E2 0.0, E3 0.0, E4 0.0, E5 0.0, E6 0.0} C_DIS
;POWDER FEED RATE  =  3.0
;LASER INTENSITY  =  4.0
LIN {E6POS: X 1462.819, Y 18.280, Z 522.849, A 43.648, B 86.259, C -136.413, E1 0.000, E2 0.0, E3 0.0, E4 0.0, E5 0.0, E6 0.0} C_DIS
;POWDER FEED RATE  =  3.0
;LASER INTENSITY  =  4.0
LIN {E6POS: X 1453.471, Y 28.440, Z 523.060, A 65.324, B 83.576, C -114.813, E1 0.000, E2 0.0, E3 0.0, E4 0.0, E5 0.0, E6 0.0} C_DIS
;POWDER FEED RATE  =  3.0
;LASER INTENSITY  =  4.0
LIN {E6POS: X 1446.188, Y 38.600, Z 524.536, A 80.693, B 74.508, C -99.651, E1 0.000, E2 0.0, E3 0.0, E4 0.0, E5 0.0, E6 0.0} C_DIS
;POWDER FEED RATE  =  3.0
;LASER INTENSITY  =  4.0
LIN {E6POS: X 1443.033, Y 48.760, Z 528.541, A 86.029, B 60.617, C -94.555, E1 0.000, E2 0.0, E3 0.0, E4 0.0, E5 0.0, E6 0.0} C_DIS
;POWDER FEED RATE  =  3.0
;LASER INTENSITY  =  4.0
LIN {E6POS: X 1445.039, Y 58.920, Z 535.708, A 87.932, B 51.371, C -92.646, E1 0.000, E2 0.0, E3 0.0, E4 0.0, E5 0.0, E6 0.0} C_DIS
;POWDER FEED RATE  =  3.0
;LASER INTENSITY  =  4.0
LIN {E6POS: X 1449.109, Y 69.080, Z 544.140, A 88.764, B 51.236, C -91.585, E1 0.000, E2 0.0, E3 0.0, E4 0.0, E5 0.0, E6 0.0} C_DIS
;POWDER FEED RATE  =  3.0
;LASER INTENSITY  =  4.0
LIN {E6POS: X 1451.115, Y 79.240, Z 551.307, A 89.195, B 60.727, C -90.923, E1 0.000, E2 0.0, E3 0.0, E4 0.0, E5 0.0, E6 0.0} C_DIS
;POWDER FEED RATE  =  3.0
;LASER INTENSITY  =  4.0
LIN {E6POS: X 1447.960, Y 89.400, Z 555.312, A 89.374, B 75.937, C -90.646, E1 0.000, E2 0.0, E3 0.0, E4 0.0, E5 0.0, E6 0.0} C_DIS
;POWDER FEED RATE  =  3.0
;LASER INTENSITY  =  4.0
LIN {E6POS: X 1440.677, Y 99.560, Z 556.788, A 89.211, B 86.396, C -90.791, E1 0.000, E2 0.0, E3 0.0, E4 0.0, E5 0.0, E6 0.0} C_DIS
;POWDER FEED RATE  =  3.0
;LASER INTENSITY  =  4.0
LIN {E6POS: X 1431.330, Y 109.720, Z 556.999, A 43.647, B 89.952, C -136.353, E1 0.000, E2 0.0, E3 0.0, E4 0.0, E5 0.0, E6 0.0} C_DIS
;POWDER FEED RATE  =  3.0
;LASER INTENSITY  =  4.0
LIN {E6POS: X 1421.639, Y 119.880, Z 556.999, A 43.647, B 89.952, C -136.353, E1 0.000, E2 0.0, E3 0.0, E4 0.0, E5 0.0, E6 0.0} C_DIS
;POWDER FEED RATE  =  3.0
;LASER INTENSITY  =  4.0
LIN {E6POS: X 1411.948, Y 130.040, Z 556.999, A 43.647, B 89.952, C -136.353, E1 0.000, E2 0.0, E3 0.0, E4 0.0, E5 0.0, E6 0.0} C_DIS
;POWDER FEED RATE  =  3.0
;LASER INTENSITY  =  4.0
LIN {E6POS: X 1402.256, Y 140.200, Z 556.999, A 43.647, B 89.952, C -136.353, E1 0.000, E2 0.0, E3 0.0, E4 0.0, E5 0.0, E6 0.0} C_DIS
;POWDER FEED RATE  =  3.0
;LASER INTENSITY  =  4.0
>>>>>>>>>>>>>>>>>>>>>>>>>>>>POWDER FEED OFF  at=START
>>>>>>>>>>>>>>>>>>>>>>>>>>>>LASER OFF at=START
>>>>>>>>>>>>>>>>>>>>>>>>>>>>GAS SUPPLY OFF  at=START
LIN {E6POS: X 1402.256, Y 140.200, Z 556.999, A 43.647, B 89.952, C -136.353, E1 0.000, E2 0.0, E3 0.0, E4 0.0, E5 0.0, E6 0.0} C_DIS
LIN {E6POS: X 1411.948, Y 130.040, Z 556.999, A 43.647, B 89.952, C -136.353, E1 0.000, E2 0.0, E3 0.0, E4 0.0, E5 0.0, E6 0.0} C_DIS
LIN {E6POS: X 1411.948, Y 130.040, Z 556.999, A 43.647, B 89.952, C -136.353, E1 0.000, E2 0.0, E3 0.0, E4 0.0, E5 0.0, E6 0.0} C_DIS
>>>>>>>>>>>>>>>>>>>>>>>>>>>>GAS SUPPLY ON at=END
>>>>>>>>>>>>>>>>>>>>>>>>>>>>POWDER FEED ON at=END
>>>>>>>>>>>>>>>>>>>>>>>>>>>>LASER ON at=END
LIN {E6POS: X 1498.375, Y -12.200, Z 523.000, A 90.000, B 90.000, C -90.000, E1 0.000, E2 0.0, E3 0.0, E4 0.0, E5 0.0, E6 0.0} C_DIS
;POWDER FEED RATE  =  3.0
;LASER INTENSITY  =  4.0
LIN {E6POS: X 1488.683, Y -2.040, Z 523.000, A 90.000, B 90.000, C -90.000, E1 0.000, E2 0.0, E3 0.0, E4 0.0, E5 0.0, E6 0.0} C_DIS
;POWDER FEED RATE  =  3.0
;LASER INTENSITY  =  4.0
LIN {E6POS: X 1478.992, Y 8.120, Z 523.000, A 90.000, B 90.000, C -90.000, E1 0.000, E2 0.0, E3 0.0, E4 0.0, E5 0.0, E6 0.0} C_DIS
;POWDER FEED RATE  =  3.0
;LASER INTENSITY  =  4.0
LIN {E6POS: X 1469.300, Y 18.280, Z 523.000, A 90.000, B 90.000, C -90.000, E1 0.000, E2 0.0, E3 0.0, E4 0.0, E5 0.0, E6 0.0} C_DIS
;POWDER FEED RATE  =  3.0
;LASER INTENSITY  =  4.0
LIN {E6POS: X 1459.954, Y 28.440, Z 523.210, A 90.000, B 86.454, C -90.000, E1 0.000, E2 0.0, E3 0.0, E4 0.0, E5 0.0, E6 0.0} C_DIS
;POWDER FEED RATE  =  3.0
;LASER INTENSITY  =  4.0
LIN {E6POS: X 1452.682, Y 38.600, Z 524.679, A 90.000, B 76.078, C -90.000, E1 0.000, E2 0.0, E3 0.0, E4 0.0, E5 0.0, E6 0.0} C_DIS
;POWDER FEED RATE  =  3.0
;LASER INTENSITY  =  4.0
LIN {E6POS: X 1449.558, Y 48.760, Z 528.667, A 90.000, B 60.850, C -90.000, E1 0.000, E2 0.0, E3 0.0, E4 0.0, E5 0.0, E6 0.0} C_DIS
;POWDER FEED RATE  =  3.0
;LASER INTENSITY  =  4.0
LIN {E6POS: X 1451.620, Y 58.920, Z 535.802, A 90.000, B 51.144, C -90.000, E1 0.000, E2 0.0, E3 0.0, E4 0.0, E5 0.0, E6 0.0} C_DIS
;POWDER FEED RATE  =  3.0
;LASER INTENSITY  =  4.0
LIN {E6POS: X 1455.755, Y 69.080, Z 544.198, A 90.000, B 51.144, C -90.000, E1 0.000, E2 0.0, E3 0.0, E4 0.0, E5 0.0, E6 0.0} C_DIS
;POWDER FEED RATE  =  3.0
;LASER INTENSITY  =  4.0
LIN {E6POS: X 1457.817, Y 79.240, Z 551.333, A 90.000, B 60.850, C -90.000, E1 0.000, E2 0.0, E3 0.0, E4 0.0, E5 0.0, E6 0.0} C_DIS
;POWDER FEED RATE  =  3.0
;LASER INTENSITY  =  4.0
LIN {E6POS: X 1454.693, Y 89.400, Z 555.321, A 90.000, B 76.078, C -90.000, E1 0.000, E2 0.0, E3 0.0, E4 0.0, E5 0.0, E6 0.0} C_DIS
;POWDER FEED RATE  =  3.0
;LASER INTENSITY  =  4.0
LIN {E6POS: X 1447.421, Y 99.560, Z 556.790, A 90.000, B 86.454, C -90.000, E1 0.000, E2 0.0, E3 0.0, E4 0.0, E5 0.0, E6 0.0} C_DIS
;POWDER FEED RATE  =  3.0
;LASER INTENSITY  =  4.0
LIN {E6POS: X 1438.075, Y 109.720, Z 557.000, A 0.000, B 90.000, C -180.000, E1 0.000, E2 0.0, E3 0.0, E4 0.0, E5 0.0, E6 0.0} C_DIS
;POWDER FEED RATE  =  3.0
;LASER INTENSITY  =  4.0
LIN {E6POS: X 1428.383, Y 119.880, Z 557.000, A 0.000, B 90.000, C -180.000, E1 0.000, E2 0.0, E3 0.0, E4 0.0, E5 0.0, E6 0.0} C_DIS
;POWDER FEED RATE  =  3.0
;LASER INTENSITY  =  4.0
LIN {E6POS: X 1418.692, Y 130.040, Z 557.000, A 0.000, B 90.000, C -180.000, E1 0.000, E2 0.0, E3 0.0, E4 0.0, E5 0.0, E6 0.0} C_DIS
;POWDER FEED RATE  =  3.0
;LASER INTENSITY  =  4.0
LIN {E6POS: X 1409.000, Y 140.200, Z 557.000, A 0.000, B 90.000, C -180.000, E1 0.000, E2 0.0, E3 0.0, E4 0.0, E5 0.0, E6 0.0} C_DIS
;POWDER FEED RATE  =  3.0
;LASER INTENSITY  =  4.0
>>>>>>>>>>>>>>>>>>>>>>>>>>>>POWDER FEED OFF  at=START
>>>>>>>>>>>>>>>>>>>>>>>>>>>>LASER OFF at=START
>>>>>>>>>>>>>>>>>>>>>>>>>>>>GAS SUPPLY OFF  at=START
LIN {E6POS: X 1409.000, Y 140.200, Z 557.000, A 0.000, B 90.000, C -180.000, E1 0.000, E2 0.0, E3 0.0, E4 0.0, E5 0.0, E6 0.0} C_DIS
LIN {E6POS: X 1418.692, Y 130.040, Z 557.000, A 0.000, B 90.000, C -180.000, E1 0.000, E2 0.0, E3 0.0, E4 0.0, E5 0.0, E6 0.0} C_DIS
LIN {E6POS: X 1418.692, Y 130.040, Z 557.000, A 0.000, B 90.000, C -180.000, E1 0.000, E2 0.0, E3 0.0, E4 0.0, E5 0.0, E6 0.0} C_DIS
>>>>>>>>>>>>>>>>>>>>>>>>>>>>GAS SUPPLY ON at=END
>>>>>>>>>>>>>>>>>>>>>>>>>>>>POWDER FEED ON at=END
>>>>>>>>>>>>>>>>>>>>>>>>>>>>LASER ON at=END
>>>>>>>>>>>>>>>>>>>>>>>>>>>>POWDER FEED OFF  at=START
>>>>>>>>>>>>>>>>>>>>>>>>>>>>GAS SUPPLY OFF  at=START
>>>>>>>>>>>>>>>>>>>>>>>>>>>>LASER OFF at=START
;FOLD ENDPOSITION PTP, VEL 50%, A1 5,A2 -90,A3 100,A4 5,A5 10,A6 -5,E1 0
$BWDSTART = FALSE
PDAT_ACT = {VEL 50,ACC 100,APO_DIST 100}
FDAT_ACT = {TOOL_NO 0,BASE_NO 0,IPO_FRAME #BASE}
BAS (#PTP_PARAMS,50)
$H_POS= {A1 5,A2 -90,A3 100,A4 5,A5 10,A6 -5,E1 0,E2 0,E3 0,E4 0,E5 0,E6 0}
PTP  {A1 5,A2 -90,A3 100,A4 5,A5 10,A6 -5,E1 0,E2 0,E3 0,E4 0,E5 0,E6 0}
;ENDFOLD
END
